INTERFACE I_Colleague

METHOD operation : BOOL
VAR_INPUT
	// Event string
	event : STRING;
END_VAR
END_METHOD

END_INTERFACE

(* stored: Version 1.1.0.1, ProductVersion 3.1.4024.12
   Itf I_Colleague: Id {0f49c02b-fca5-4a43-8d8f-e44ce45a3e83}
   Method operation: Id {df911ca8-2d22-4547-bcd9-63adfb09aa95} *)
